(* Logix 5000 project; controller cal1632 1756-L62 rev 16.20; software revision 16.05; part 12 of 61 *)
(* tags used below, declared in another part *)
   FAULT : BOOL;
   HMI : BOOL;
   p01r09_pb_global_reset : BOOL;
   p11_ai_exh_amps : REAL;
   p11_ai_exh_hz : REAL;
   p11_ai_exh_pct : REAL;
   p11_ai_exh_rpm : REAL;
   p11_ai_lfl : REAL;
   p11_ai_prs : REAL;
   p11_ai_recirc_amps : REAL;
   p11_ai_recirc_hz : REAL;
   p11_ai_recirc_pct : REAL;
   p11_ai_recirc_rpm : REAL;
   p11_ai_tc01 : REAL;
   p11_ai_tc02 : REAL;
   p11_ao_cv : REAL;
   p11_ao_exhaust_selected_speed : REAL;
   p11_ao_recirc_selected_speed : REAL;
   p11_dint_to_hmi : DINT[16];
   p11_param_fast_to_soak : REAL;
   p11_param_lfl_hhl : REAL;
   p11_param_lfl_hl : REAL;
   p11_param_pid1_ff : REAL;
   p11_param_pid1_kd : REAL;
   p11_param_pid1_ki : REAL;
   p11_param_pid1_kp : REAL;
   p11_param_pid2_ff : REAL;
   p11_param_pid2_kd : REAL;
   p11_param_pid2_ki : REAL;
   p11_param_pid2_kp : REAL;
   p11_param_shutdown_temp : REAL;
   p11_param_soak_to_fast : REAL;
   p11_param_tc01_dev : REAL;
   p11_param_tc01_hl : REAL;
   p11_param_tc01z : REAL;
   p11_param_tc02z : REAL;
   p11_param_zone_pressure : REAL;
   p11_real_to_hmi : REAL[112];
   p11r02 : routine;
   p11r06 : routine;
   p11r06_timer_fault : TIMER[4];
   p11r06_timer_warning : TIMER[4];
   p11r07 : routine;
   p11r07_timer_fault : TIMER[4];
   p11r07_timer_warning : TIMER[4];
   p11r08 : routine;
   p11r08_timer_fault : TIMER[4];
   p11r08_timer_warning : TIMER[4];
   p11r09 : routine;
   p11r09_timer_fault : TIMER[4];
   p11r09_timer_warning : TIMER[8];
   p11r20 : routine;
   p11r30 : routine;
   p11r30_cv_man_sp : REAL;
   p11r30_pid_temp : PID;
   p11r30_pid_temp_pv : REAL;
   p11r30_pid_temp_sp : REAL;
   p11r31 : routine;
   p11r32 : routine;
(* P11_Zone_1, continued *)

ROUTINE R06_Real_to_HMI   (* ladder *)
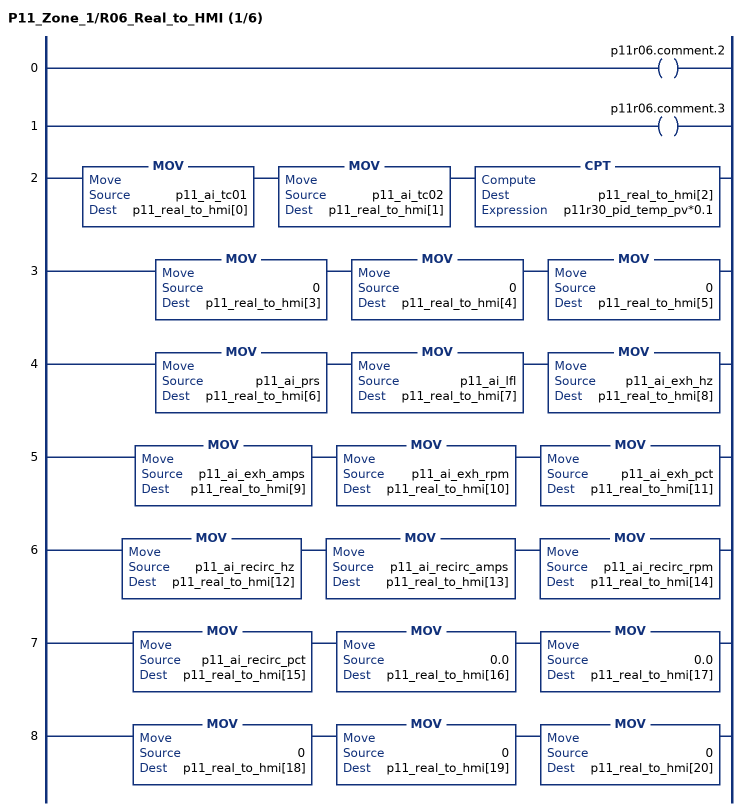
   0: OTE(p11r06.comment.2);
   1: OTE(p11r06.comment.3);
   2: MOV(p11_ai_tc01,p11_real_to_hmi[0])MOV(p11_ai_tc02,p11_real_to_hmi[1])CPT(p11_real_to_hmi[2],p11r30_pid_temp_pv*0.1);
   3: MOV(0,p11_real_to_hmi[3])MOV(0,p11_real_to_hmi[4])MOV(0,p11_real_to_hmi[5]);
   4: MOV(p11_ai_prs,p11_real_to_hmi[6])MOV(p11_ai_lfl,p11_real_to_hmi[7])MOV(p11_ai_exh_hz,p11_real_to_hmi[8]);
   5: MOV(p11_ai_exh_amps,p11_real_to_hmi[9])MOV(p11_ai_exh_rpm,p11_real_to_hmi[10])MOV(p11_ai_exh_pct,p11_real_to_hmi[11]);
   6: MOV(p11_ai_recirc_hz,p11_real_to_hmi[12])MOV(p11_ai_recirc_amps,p11_real_to_hmi[13])MOV(p11_ai_recirc_rpm,p11_real_to_hmi[14]);
   7: MOV(p11_ai_recirc_pct,p11_real_to_hmi[15])MOV(0.0,p11_real_to_hmi[16])MOV(0.0,p11_real_to_hmi[17]);
   8: MOV(0,p11_real_to_hmi[18])MOV(0,p11_real_to_hmi[19])MOV(0,p11_real_to_hmi[20]);
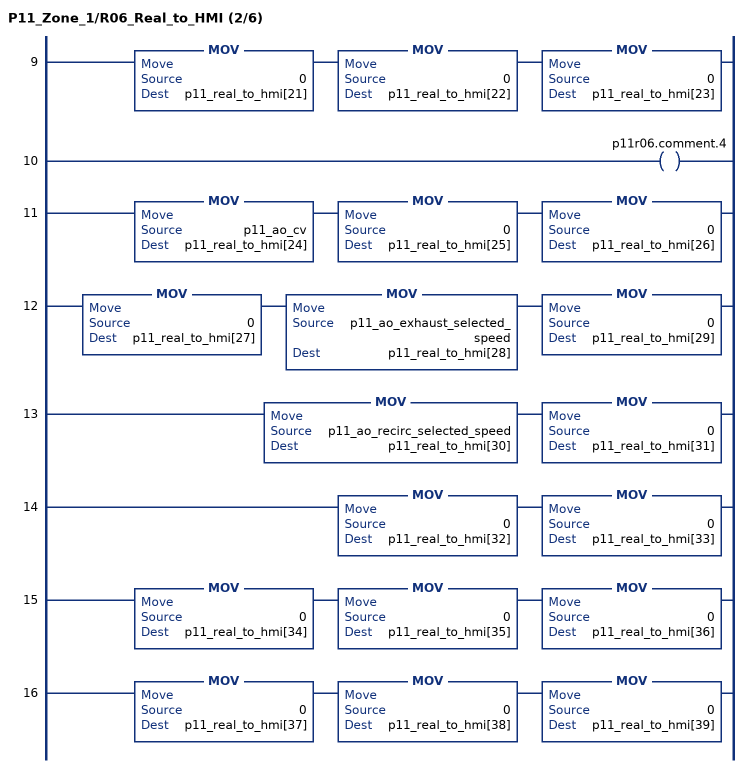
   9: MOV(0,p11_real_to_hmi[21])MOV(0,p11_real_to_hmi[22])MOV(0,p11_real_to_hmi[23]);
   10: OTE(p11r06.comment.4);
   11: MOV(p11_ao_cv,p11_real_to_hmi[24])MOV(0,p11_real_to_hmi[25])MOV(0,p11_real_to_hmi[26]);
   12: MOV(0,p11_real_to_hmi[27])MOV(p11_ao_exhaust_selected_speed,p11_real_to_hmi[28])MOV(0,p11_real_to_hmi[29]);
   13: MOV(p11_ao_recirc_selected_speed,p11_real_to_hmi[30])MOV(0,p11_real_to_hmi[31]);
   14: MOV(0,p11_real_to_hmi[32])MOV(0,p11_real_to_hmi[33]);
   15: MOV(0,p11_real_to_hmi[34])MOV(0,p11_real_to_hmi[35])MOV(0,p11_real_to_hmi[36]);
   16: MOV(0,p11_real_to_hmi[37])MOV(0,p11_real_to_hmi[38])MOV(0,p11_real_to_hmi[39]);
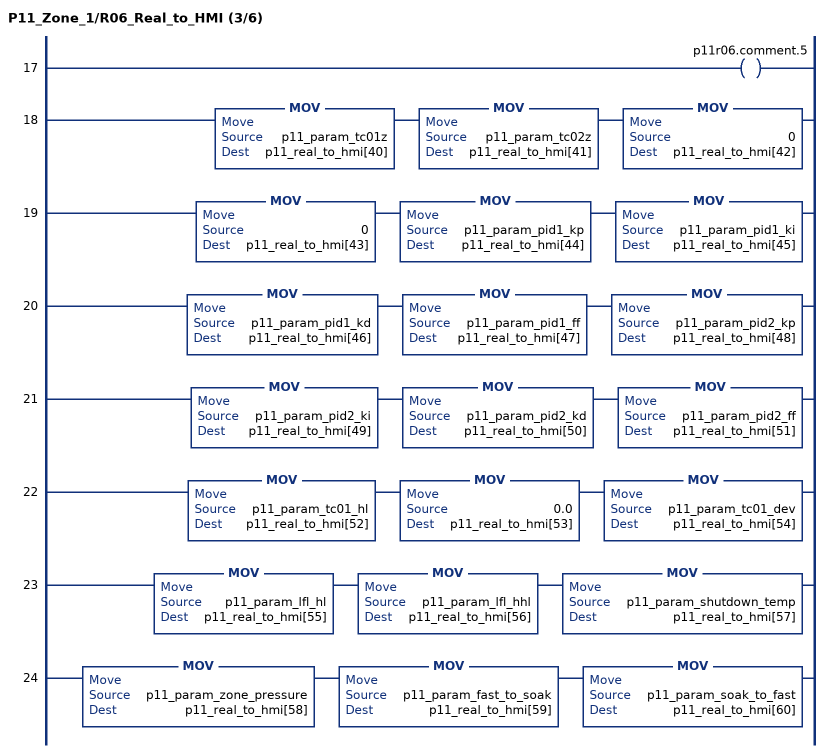
   17: OTE(p11r06.comment.5);
   18: MOV(p11_param_tc01z,p11_real_to_hmi[40])MOV(p11_param_tc02z,p11_real_to_hmi[41])MOV(0,p11_real_to_hmi[42]);
   19: MOV(0,p11_real_to_hmi[43])MOV(p11_param_pid1_kp,p11_real_to_hmi[44])MOV(p11_param_pid1_ki,p11_real_to_hmi[45]);
   20: MOV(p11_param_pid1_kd,p11_real_to_hmi[46])MOV(p11_param_pid1_ff,p11_real_to_hmi[47])MOV(p11_param_pid2_kp,p11_real_to_hmi[48]);
   21: MOV(p11_param_pid2_ki,p11_real_to_hmi[49])MOV(p11_param_pid2_kd,p11_real_to_hmi[50])MOV(p11_param_pid2_ff,p11_real_to_hmi[51]);
   22: MOV(p11_param_tc01_hl,p11_real_to_hmi[52])MOV(0.0,p11_real_to_hmi[53])MOV(p11_param_tc01_dev,p11_real_to_hmi[54]);
   23: MOV(p11_param_lfl_hl,p11_real_to_hmi[55])MOV(p11_param_lfl_hhl,p11_real_to_hmi[56])MOV(p11_param_shutdown_temp,p11_real_to_hmi[57]);
   24: MOV(p11_param_zone_pressure,p11_real_to_hmi[58])MOV(p11_param_fast_to_soak,p11_real_to_hmi[59])MOV(p11_param_soak_to_fast,p11_real_to_hmi[60]);
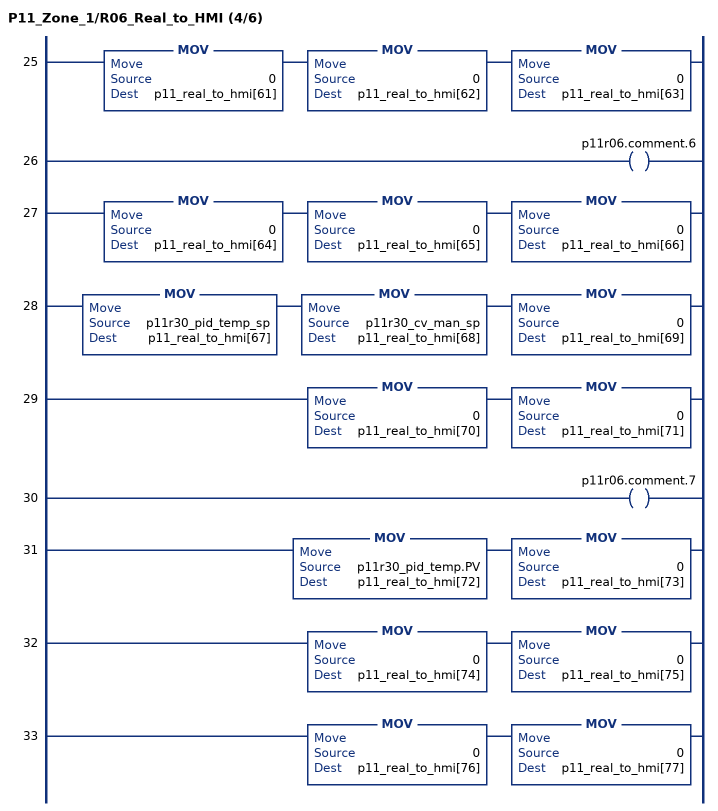
   25: MOV(0,p11_real_to_hmi[61])MOV(0,p11_real_to_hmi[62])MOV(0,p11_real_to_hmi[63]);
   26: OTE(p11r06.comment.6);
   27: MOV(0,p11_real_to_hmi[64])MOV(0,p11_real_to_hmi[65])MOV(0,p11_real_to_hmi[66]);
   28: MOV(p11r30_pid_temp_sp,p11_real_to_hmi[67])MOV(p11r30_cv_man_sp,p11_real_to_hmi[68])MOV(0,p11_real_to_hmi[69]);
   29: MOV(0,p11_real_to_hmi[70])MOV(0,p11_real_to_hmi[71]);
   30: OTE(p11r06.comment.7);
   31: MOV(p11r30_pid_temp.PV,p11_real_to_hmi[72])MOV(0,p11_real_to_hmi[73]);
   32: MOV(0,p11_real_to_hmi[74])MOV(0,p11_real_to_hmi[75]);
   33: MOV(0,p11_real_to_hmi[76])MOV(0,p11_real_to_hmi[77]);
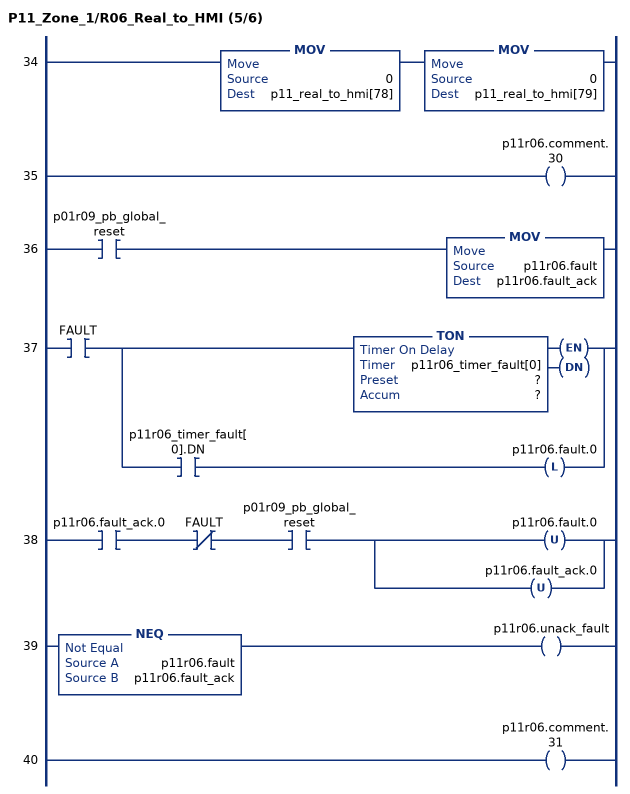
   34: MOV(0,p11_real_to_hmi[78])MOV(0,p11_real_to_hmi[79]);
   35: OTE(p11r06.comment.30);
   36: XIC(p01r09_pb_global_reset)MOV(p11r06.fault,p11r06.fault_ack);
   37: XIC(FAULT)[TON(p11r06_timer_fault[0],?,?) ,XIC(p11r06_timer_fault[0].DN) OTL(p11r06.fault.0) ];
   38: XIC(p11r06.fault_ack.0)XIO(FAULT)XIC(p01r09_pb_global_reset)[OTU(p11r06.fault.0) ,OTU(p11r06.fault_ack.0) ];
   39: NEQ(p11r06.fault,p11r06.fault_ack)OTE(p11r06.unack_fault);
   40: OTE(p11r06.comment.31);
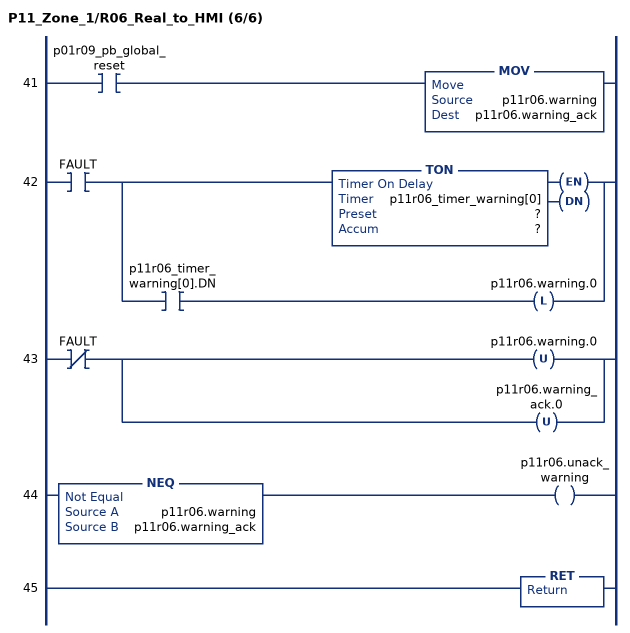
   41: XIC(p01r09_pb_global_reset)MOV(p11r06.warning,p11r06.warning_ack);
   42: XIC(FAULT)[TON(p11r06_timer_warning[0],?,?) ,XIC(p11r06_timer_warning[0].DN) OTL(p11r06.warning.0) ];
   43: XIO(FAULT)[OTU(p11r06.warning.0) ,OTU(p11r06.warning_ack.0) ];
   44: NEQ(p11r06.warning,p11r06.warning_ack)OTE(p11r06.unack_warning);
   45: RET();
END_ROUTINE

ROUTINE R07_Alarms   (* ladder *)
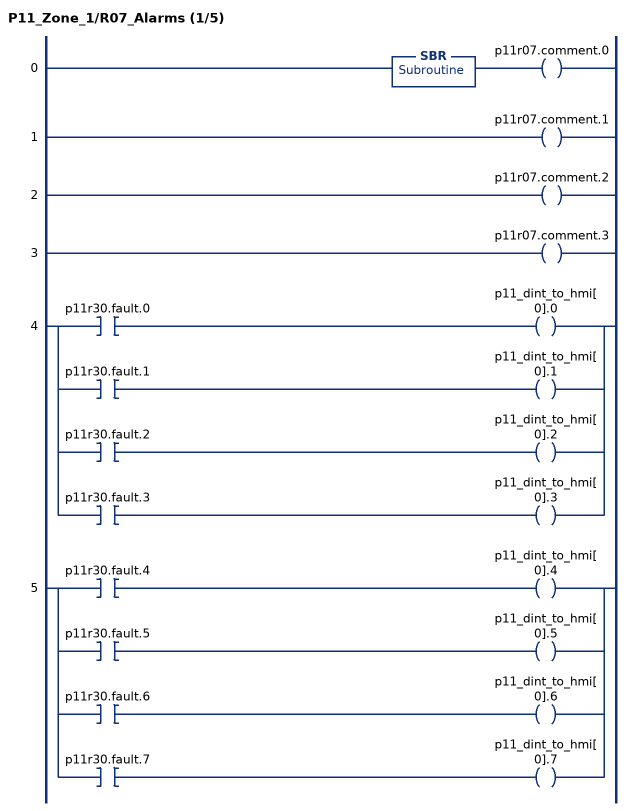
   0: SBR()OTE(p11r07.comment.0);
   1: OTE(p11r07.comment.1);
   2: OTE(p11r07.comment.2);
   3: OTE(p11r07.comment.3);
   4: [XIC(p11r30.fault.0) OTE(p11_dint_to_hmi[0].0) ,XIC(p11r30.fault.1) OTE(p11_dint_to_hmi[0].1) ,XIC(p11r30.fault.2) OTE(p11_dint_to_hmi[0].2) ,XIC(p11r30.fault.3) OTE(p11_dint_to_hmi[0].3) ];
   5: [XIC(p11r30.fault.4) OTE(p11_dint_to_hmi[0].4) ,XIC(p11r30.fault.5) OTE(p11_dint_to_hmi[0].5) ,XIC(p11r30.fault.6) OTE(p11_dint_to_hmi[0].6) ,XIC(p11r30.fault.7) OTE(p11_dint_to_hmi[0].7) ];
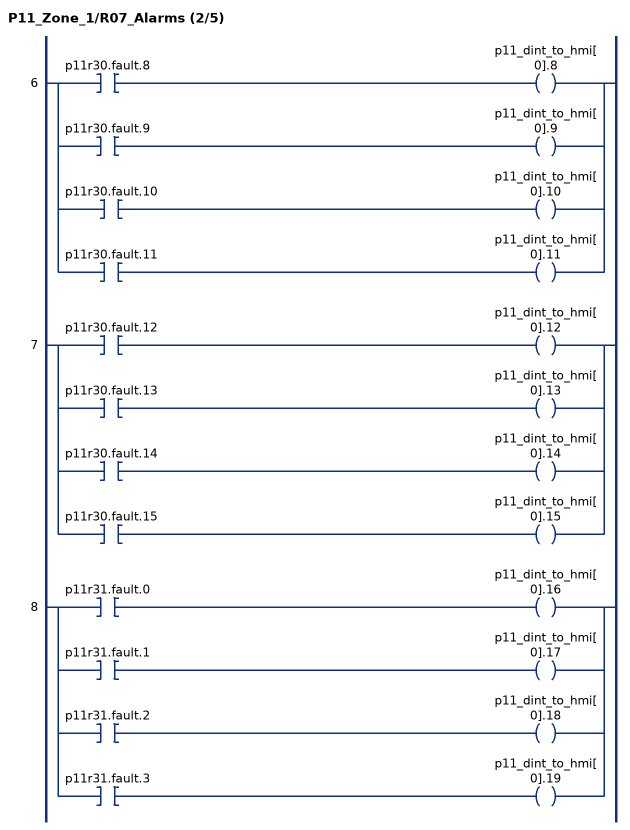
   6: [XIC(p11r30.fault.8) OTE(p11_dint_to_hmi[0].8) ,XIC(p11r30.fault.9) OTE(p11_dint_to_hmi[0].9) ,XIC(p11r30.fault.10) OTE(p11_dint_to_hmi[0].10) ,XIC(p11r30.fault.11) OTE(p11_dint_to_hmi[0].11) ];
   7: [XIC(p11r30.fault.12) OTE(p11_dint_to_hmi[0].12) ,XIC(p11r30.fault.13) OTE(p11_dint_to_hmi[0].13) ,XIC(p11r30.fault.14) OTE(p11_dint_to_hmi[0].14) ,XIC(p11r30.fault.15) OTE(p11_dint_to_hmi[0].15) ];
   8: [XIC(p11r31.fault.0) OTE(p11_dint_to_hmi[0].16) ,XIC(p11r31.fault.1) OTE(p11_dint_to_hmi[0].17) ,XIC(p11r31.fault.2) OTE(p11_dint_to_hmi[0].18) ,XIC(p11r31.fault.3) OTE(p11_dint_to_hmi[0].19) ];
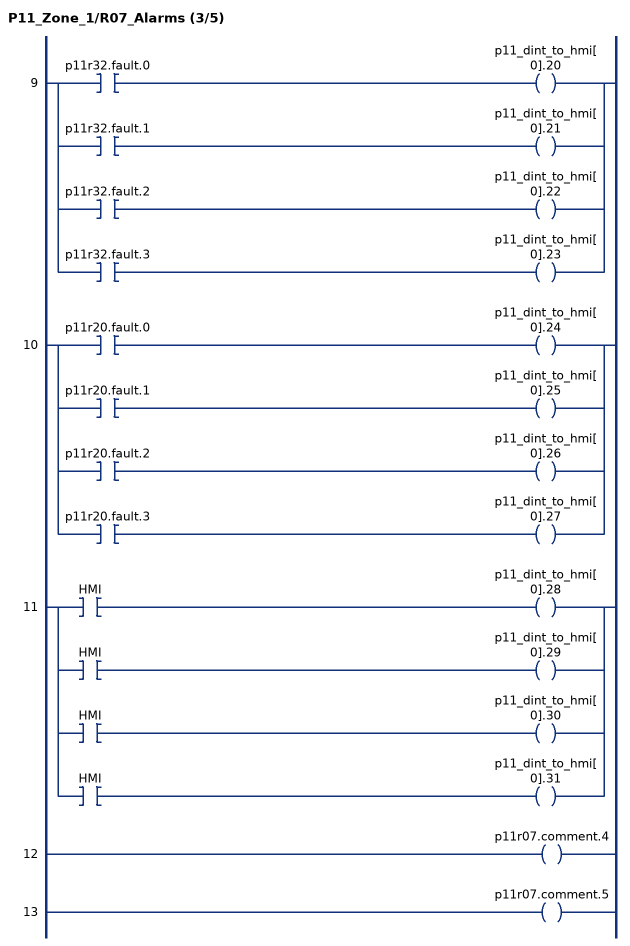
   9: [XIC(p11r32.fault.0) OTE(p11_dint_to_hmi[0].20) ,XIC(p11r32.fault.1) OTE(p11_dint_to_hmi[0].21) ,XIC(p11r32.fault.2) OTE(p11_dint_to_hmi[0].22) ,XIC(p11r32.fault.3) OTE(p11_dint_to_hmi[0].23) ];
   10: [XIC(p11r20.fault.0) OTE(p11_dint_to_hmi[0].24) ,XIC(p11r20.fault.1) OTE(p11_dint_to_hmi[0].25) ,XIC(p11r20.fault.2) OTE(p11_dint_to_hmi[0].26) ,XIC(p11r20.fault.3) OTE(p11_dint_to_hmi[0].27) ];
   11: [XIC(HMI) OTE(p11_dint_to_hmi[0].28) ,XIC(HMI) OTE(p11_dint_to_hmi[0].29) ,XIC(HMI) OTE(p11_dint_to_hmi[0].30) ,XIC(HMI) OTE(p11_dint_to_hmi[0].31) ];
   12: OTE(p11r07.comment.4);
   13: OTE(p11r07.comment.5);
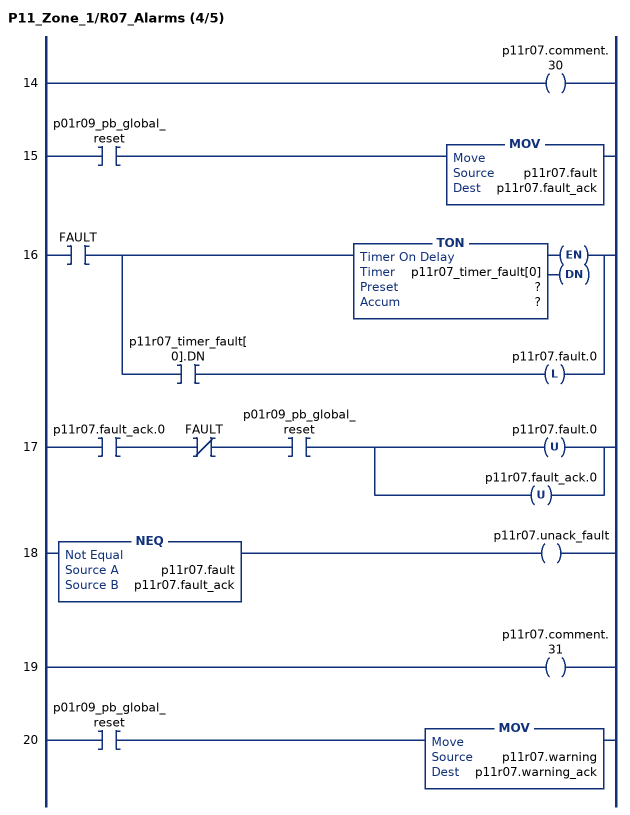
   14: OTE(p11r07.comment.30);
   15: XIC(p01r09_pb_global_reset)MOV(p11r07.fault,p11r07.fault_ack);
   16: XIC(FAULT)[TON(p11r07_timer_fault[0],?,?) ,XIC(p11r07_timer_fault[0].DN) OTL(p11r07.fault.0) ];
   17: XIC(p11r07.fault_ack.0)XIO(FAULT)XIC(p01r09_pb_global_reset)[OTU(p11r07.fault.0) ,OTU(p11r07.fault_ack.0) ];
   18: NEQ(p11r07.fault,p11r07.fault_ack)OTE(p11r07.unack_fault);
   19: OTE(p11r07.comment.31);
   20: XIC(p01r09_pb_global_reset)MOV(p11r07.warning,p11r07.warning_ack);
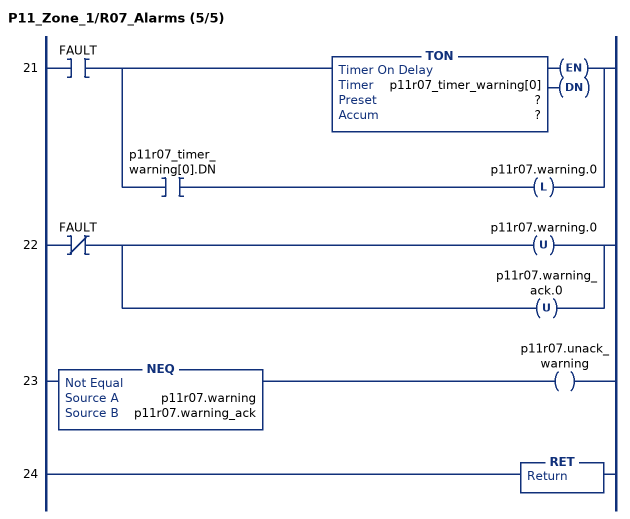
   21: XIC(FAULT)[TON(p11r07_timer_warning[0],?,?) ,XIC(p11r07_timer_warning[0].DN) OTL(p11r07.warning.0) ];
   22: XIO(FAULT)[OTU(p11r07.warning.0) ,OTU(p11r07.warning_ack.0) ];
   23: NEQ(p11r07.warning,p11r07.warning_ack)OTE(p11r07.unack_warning);
   24: RET();
END_ROUTINE

ROUTINE R08_Warnings   (* ladder *)
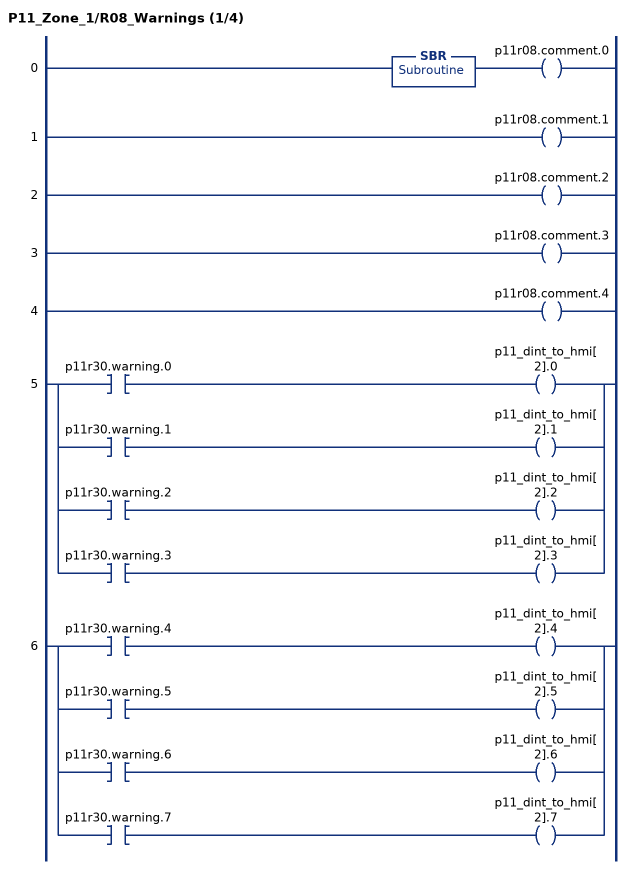
   0: SBR()OTE(p11r08.comment.0);
   1: OTE(p11r08.comment.1);
   2: OTE(p11r08.comment.2);
   3: OTE(p11r08.comment.3);
   4: OTE(p11r08.comment.4);
   5: [XIC(p11r30.warning.0) OTE(p11_dint_to_hmi[2].0) ,XIC(p11r30.warning.1) OTE(p11_dint_to_hmi[2].1) ,XIC(p11r30.warning.2) OTE(p11_dint_to_hmi[2].2) ,XIC(p11r30.warning.3) OTE(p11_dint_to_hmi[2].3) ];
   6: [XIC(p11r30.warning.4) OTE(p11_dint_to_hmi[2].4) ,XIC(p11r30.warning.5) OTE(p11_dint_to_hmi[2].5) ,XIC(p11r30.warning.6) OTE(p11_dint_to_hmi[2].6) ,XIC(p11r30.warning.7) OTE(p11_dint_to_hmi[2].7) ];
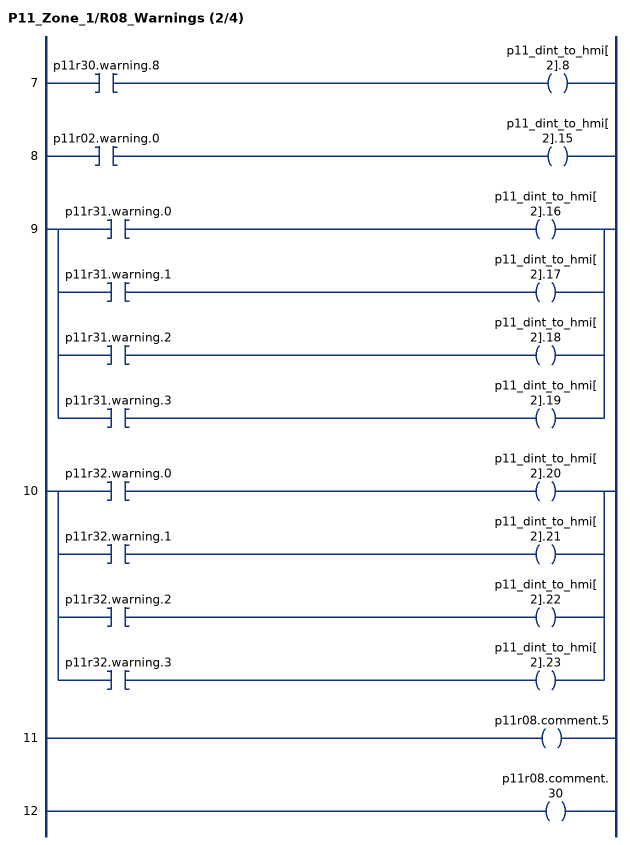
   7: XIC(p11r30.warning.8)OTE(p11_dint_to_hmi[2].8);
   8: XIC(p11r02.warning.0)OTE(p11_dint_to_hmi[2].15);
   9: [XIC(p11r31.warning.0) OTE(p11_dint_to_hmi[2].16) ,XIC(p11r31.warning.1) OTE(p11_dint_to_hmi[2].17) ,XIC(p11r31.warning.2) OTE(p11_dint_to_hmi[2].18) ,XIC(p11r31.warning.3) OTE(p11_dint_to_hmi[2].19) ];
   10: [XIC(p11r32.warning.0) OTE(p11_dint_to_hmi[2].20) ,XIC(p11r32.warning.1) OTE(p11_dint_to_hmi[2].21) ,XIC(p11r32.warning.2) OTE(p11_dint_to_hmi[2].22) ,XIC(p11r32.warning.3) OTE(p11_dint_to_hmi[2].23) ];
   11: OTE(p11r08.comment.5);
   12: OTE(p11r08.comment.30);
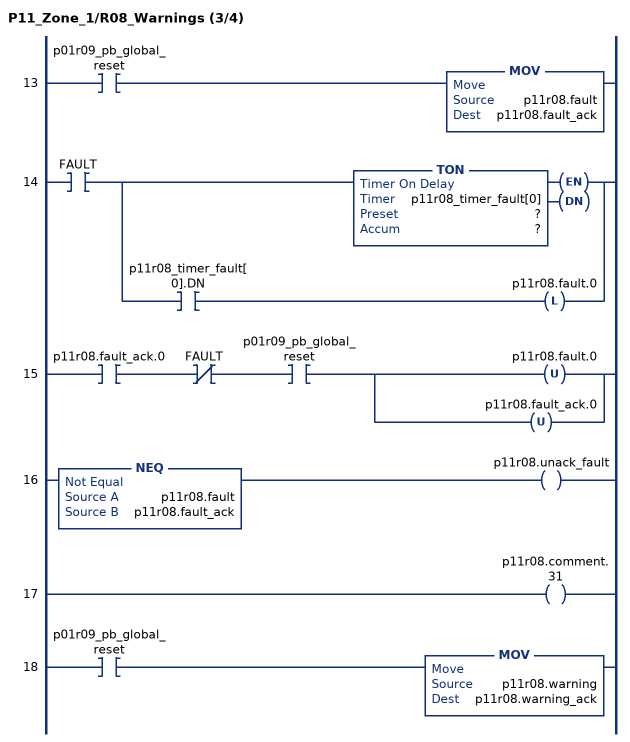
   13: XIC(p01r09_pb_global_reset)MOV(p11r08.fault,p11r08.fault_ack);
   14: XIC(FAULT)[TON(p11r08_timer_fault[0],?,?) ,XIC(p11r08_timer_fault[0].DN) OTL(p11r08.fault.0) ];
   15: XIC(p11r08.fault_ack.0)XIO(FAULT)XIC(p01r09_pb_global_reset)[OTU(p11r08.fault.0) ,OTU(p11r08.fault_ack.0) ];
   16: NEQ(p11r08.fault,p11r08.fault_ack)OTE(p11r08.unack_fault);
   17: OTE(p11r08.comment.31);
   18: XIC(p01r09_pb_global_reset)MOV(p11r08.warning,p11r08.warning_ack);
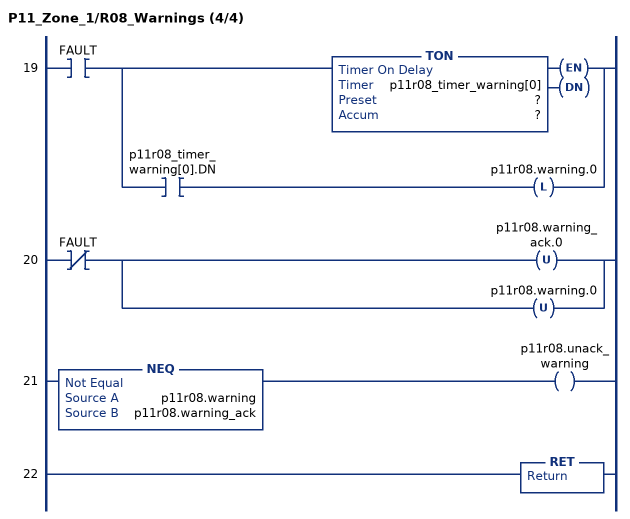
   19: XIC(FAULT)[TON(p11r08_timer_warning[0],?,?) ,XIC(p11r08_timer_warning[0].DN) OTL(p11r08.warning.0) ];
   20: XIO(FAULT)[OTU(p11r08.warning_ack.0) ,OTU(p11r08.warning.0) ];
   21: NEQ(p11r08.warning,p11r08.warning_ack)OTE(p11r08.unack_warning);
   22: RET();
END_ROUTINE

ROUTINE R09_Modes   (* ladder *)
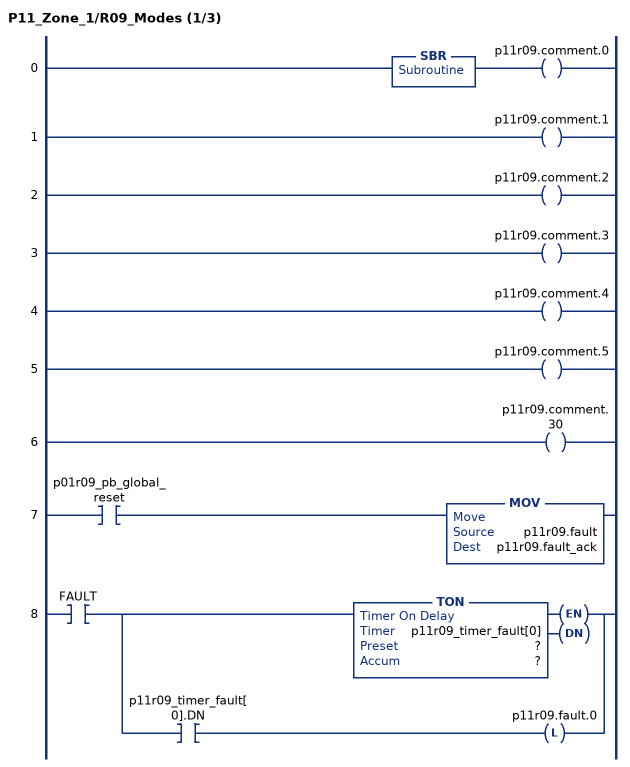
   0: SBR()OTE(p11r09.comment.0);
   1: OTE(p11r09.comment.1);
   2: OTE(p11r09.comment.2);
   3: OTE(p11r09.comment.3);
   4: OTE(p11r09.comment.4);
   5: OTE(p11r09.comment.5);
   6: OTE(p11r09.comment.30);
   7: XIC(p01r09_pb_global_reset)MOV(p11r09.fault,p11r09.fault_ack);
   8: XIC(FAULT)[TON(p11r09_timer_fault[0],?,?) ,XIC(p11r09_timer_fault[0].DN) OTL(p11r09.fault.0) ];
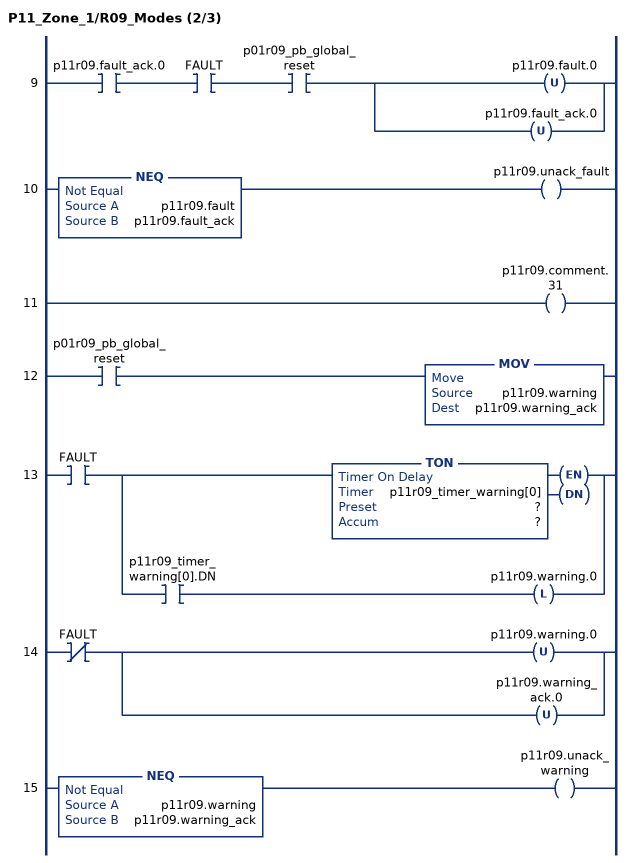
   9: XIC(p11r09.fault_ack.0)XIC(FAULT)XIC(p01r09_pb_global_reset)[OTU(p11r09.fault.0) ,OTU(p11r09.fault_ack.0) ];
   10: NEQ(p11r09.fault,p11r09.fault_ack)OTE(p11r09.unack_fault);
   11: OTE(p11r09.comment.31);
   12: XIC(p01r09_pb_global_reset)MOV(p11r09.warning,p11r09.warning_ack);
   13: XIC(FAULT)[TON(p11r09_timer_warning[0],?,?) ,XIC(p11r09_timer_warning[0].DN) OTL(p11r09.warning.0) ];
   14: XIO(FAULT)[OTU(p11r09.warning.0) ,OTU(p11r09.warning_ack.0) ];
   15: NEQ(p11r09.warning,p11r09.warning_ack)OTE(p11r09.unack_warning);
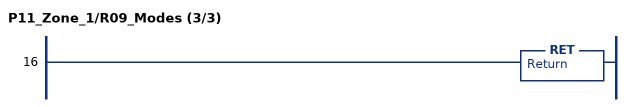
   16: RET();
END_ROUTINE
